Fanuc KAREL source: kd00008.KL

-- PROVISIONAL review KL for V770-1; original PC SHA256 7233dc1da045fca2325eb42d25e2f719eaf66b91daec5e7febf786c103a0407d
-- Incomplete behavior may be omitted. Consult companion uncertainty JSON. Do not deploy.
PROGRAM KD00008
%NOLOCKGROUP
VAR
  I : INTEGER
  J : INTEGER
  B : BOOLEAN
  R : REAL
  S : STRING[80]
BEGIN
  -- UNRESOLVED_PC offsets 5-12; opcodes 9D,23
  -- UNRESOLVED_PC offsets 17-21; opcodes 7F
END KD00008
